// TIA Portal V16 export
// export: Created 2024-12-03T15:41:45.5327184Z, ExportSetting WithReadOnly, DisplayName Totally Integrated Automation Portal, DisplayVersion V16 Update 6, DisplayName TIA Portal Version Control Interface, DisplayVersion V16 Update 2, DisplayName TIA Portal Openness, DisplayVersion V16 Update 6, DisplayName TIA Portal Teamcenter Gateway, DisplayVersion V16, DisplayName SINAMICS Startdrive Advanced, DisplayVersion V16 Update 5, DisplayName SINAMICS Startdrive G130, G150, S120, S150, SINAMICS MV, S210, DisplayVersion V16 Update 5, DisplayName SINAMICS Startdrive G110M, G120, G120C, G120D, G120P, G115D, DisplayVersion V16 Update 5, DisplayName STEP 7 Professional, DisplayVersion V16 Update 6, DisplayName STEP 7 Safety, DisplayVersion V16, DisplayName WinCC Advanced / Unified PC, DisplayVersion V16 Update 6
TYPE "I_RANPACK_UDT"
// stored: CreationDate 2022-02-11T09:59:07.2809667Z, InterfaceModifiedDate 2022-02-11T10:07:18.2853623Z, IsConsistent true, LibraryConformanceStatus The object is library-conformant., ModifiedDate 2022-02-11T10:07:18.2853623Z
   STRUCT
      status : Struct
         readyToReceive : Bool;
         readyToSent : Bool;
         machineError : Bool;
         spare : Bool;
         lidSupplyLowWarning : Bool;
         GlueSupplyLowWarning : Bool;
         LidSupplyLowError : Bool;
         GlueSupplyLowError : Bool;
         spare_1 : Bool;
         spare_2 : Bool;
         spare_3 : Bool;
         spare_4 : Bool;
         spare_5 : Bool;
         TransferInProgress : Bool;
         DataReceived : Bool;
         KeepAlive : Bool;
      END_STRUCT;
      ObjectInfo : Struct
         CuttingError : Bool;
         LiddingError : Bool;
         CuttingOk : Bool;
         WithoutCutting : Bool;
         withoutLidding : Bool;
         spare : Bool;
         spare_1 : Bool;
         spare_2 : Bool;
         Barcode_1 : Char;
         Barcode_2 : Char;
         Barcode_3 : Char;
         Barcode_4 : Char;
         Barcode_5 : Char;
         Barcode_6 : Char;
         Barcode_7 : Char;
         Barcode_8 : Char;
         Barcode_9 : Char;
         Barcode_10 : Char;
         Barcode_11 : Char;
         Barcode_12 : Char;
         Barcode_13 : Char;
         Barcode_14 : Char;
         Barcode_15 : Char;
         Barcode_16 : Char;
         weight : Byte;   // Weight in KG
         Length : Word;
         widht : Word;
         HeightBoxBasis : Word;
         HeightBoxProduct : Word;
         HeightBoxFinel : Word;
         HeightBoxMinimum : Byte;
         MinimumCut : Byte;
      END_STRUCT;
   END_STRUCT;
END_TYPE
